FUNCTION_BLOCK FB_MainHMI_Connection
VAR_IN_OUT
END_VAR
VAR_INPUT
	sTopLevelMachine : STRING;
END_VAR
VAR_OUTPUT
END_VAR
VAR
	fbModuleTree : FB_Tree_IndexBased;
	a_stMachineTreeNodes	: ARRAY[0..63] OF ST_Tree_IndexBased_Node;
	bInitialized : BOOL;

END_VAR

IF NOT bInitialized THEN
	(*
	sTopLevelMachine := 'My machine';		//TODO: Proper implementation of auto-generating tree structure
	fbModuleTree(a_stNodes := stMachineTreeNodes, sHead := sTopLevelMachine);
	fbModuleTree.AddNodeAsChildByName(sNewName := 'EM1', sParentName := 'My machine');
	fbModuleTree.AddNodeAsChildByName(sNewName := 'CM1', sParentName := 'EM1');
	fbModuleTree.AddNodeAsChildByName(sNewName := 'CP1', sParentName := 'CM1');
	fbModuleTree.AddNodeAsChildByName(sNewName := 'CP2', sParentName := 'CM1');
	fbModuleTree.AddNodeAsChildByName(sNewName := 'CM2', sParentName := 'EM1');
	fbModuleTree.AddNodeAsChildByName(sNewName := 'CM3', sParentName := 'EM1');
	fbModuleTree.AddNodeAsChildByName(sNewName := 'CP3', sParentName := 'CM3');
	fbModuleTree.AddNodeAsChildByName(sNewName := 'EM2', sParentName := 'My machine');
	fbModuleTree.AddNodeAsChildByName(sNewName := 'CM4', sParentName := 'EM2');
	fbModuleTree.AddNodeAsChildByName(sNewName := 'CM5', sParentName := 'EM2');
	fbModuleTree.AddNodeAsChildByName(sNewName := 'CP4', sParentName := 'CM5');
	fbModuleTree.AddNodeAsChildByName(sNewName := 'CP5', sParentName := 'CM5');
	fbModuleTree.AddNodeAsChildByName(sNewName := 'CP10', sParentName := 'CM5');
	fbModuleTree.AddNodeAsChildByName(sNewName := 'CP11', sParentName := 'CM5');
	fbModuleTree.AddNodeAsChildByName(sNewName := 'CP12', sParentName := 'CM5');
	fbModuleTree.AddNodeAsChildByName(sNewName := 'CM6', sParentName := 'EM2');
	fbModuleTree.AddNodeAsChildByName(sNewName := 'CM7', sParentName := 'EM2');
	fbModuleTree.AddNodeAsChildByName(sNewName := 'CP7', sParentName := 'CM7');
	fbModuleTree.AddNodeAsChildByName(sNewName := 'EM3', sParentName := 'My machine');
	fbModuleTree.AddNodeAsChildByName(sNewName := 'CM8', sParentName := 'EM3');
	fbModuleTree.AddNodeAsChildByName(sNewName := 'CM9', sParentName := 'EM3');
	fbModuleTree.AddNodeAsChildByName(sNewName := 'CP8', sParentName := 'CM9');
	fbModuleTree.AddNodeAsChildByName(sNewName := 'CP9', sParentName := 'CM9');
	fbModuleTree.AddNodeAsChildByName(sNewName := 'EM4', sParentName := 'My machine');
	*)
	fbModuleTree(a_stNodes := a_stMachineTreeNodes, sHead := sTopLevelMachine);
	
	bInitialized := TRUE;
END_IF

PROPERTY DataStructure_Adder : ITF_Tree_IndexBased
GET
DataStructure_Adder := fbModuleTree;
END_GET
END_PROPERTY

END_FUNCTION_BLOCK

(* stored: Version 1.1.0.1, ProductVersion 3.1.4024.10
   POU FB_MainHMI_Connection: Id {c1188b0b-fda8-400d-83a0-4bed5c564a86}, SpecialFunc None
   Property DataStructure_Adder: Id {acd045ca-4fdd-4391-9486-4c599ce99025}
   Get Get: Id {7fccfe0b-bcf0-439a-b53c-58c304b9527a} *)
